SUBAPPLICATION mapping (* Subapplication Type *)
  (* Standard: 61499-2 *)
  (* Version 1.0, 2024-03-23, franz *)
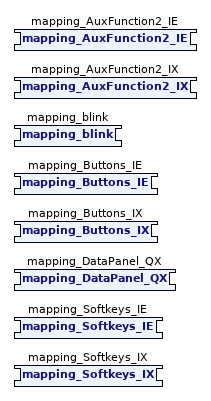
  SUBAPPS
    mapping_AuxFunction2_IE : mapping_AuxFunction2_IE;
    mapping_AuxFunction2_IX : mapping_AuxFunction2_IX;
    mapping_blink : mapping_blink;
    mapping_Buttons_IE : mapping_Buttons_IE;
    mapping_Buttons_IX : mapping_Buttons_IX;
    mapping_DataPanel_QX : mapping_DataPanel_QX;
    mapping_Softkeys_IE : mapping_Softkeys_IE;
    mapping_Softkeys_IX : mapping_Softkeys_IX;
  END_SUBAPPS
END_SUBAPPLICATION
